FUNCTION WRITE_ANY_DWORD : BOOL
VAR_INPUT
    ptr: POINTER TO DWORD;
    val: DWORD;
END_VAR

ptr^ := val;

END_FUNCTION

(* stored: Version 1.1.0.1, ProductVersion 3.1.4022.9
   POU WRITE_ANY_DWORD: Id {adb6e532-53d2-41dc-9582-b0d035315f3a}, SpecialFunc None *)
